PROGRAM CAN_comm
VAR
	i : INT := 0; // data 0 - 7 
	j : INT := 1; // coil 1-10
	k : INT := 1; // uc 1-10
	
	hmi_sendRequest : BOOL;
	hmi_step1 : BOOL;
	hmi_step2 : BOOL;
	hmi_step3 : BOOL;
	hmi_step4 : BOOL;
	hmi_step5 : BOOL;
	//hmi_CanTxB_str	: ARRAY [0..7] OF STRING;
	//hmi_CanTxB		: ARRAY [0..7] OF BYTE;
	hmi_CanTx_ID_str	: STRING;
	hmi_CanTx_ID		: UDINT;
	//hmi_CanTx_length	: UINT;
	hmi_CanTx_desiredID : STRING;
	hmi_CanTx_desID		: BYTE;

END_VAR

//0x0CF091 XX ELECTRICAL DATA
//0x0CF092 XX THERMAL DATA

//XX 
// ie 0x11[overvoltage][imbalance][blancing]
//data[0] = Electrical flag | data[1], data[2] = Voltage sum | data[3], data[4] = highest voltage | data[5], data[6] = average voltage | data[7] = life counter
//data[0].0
//data[0].1  Balancing
//data[0].2  
//data[0].3  Imbalance
//data[0].4
//data[0].5  Overvoltage
//data[0].6 = 1
//data[0].7 = 1

Devices.Coil[j].UC_Dummy_ID_hexstr :=  (DWORD_TO_HEXSTR (in := Devices.Coil[j].UltraCap_Dummy.R2_06_UC_Rx_cobID, iPrecision := 2, bLoCase := FALSE));
	//Devices.Coil[1].UltraCap_CAN_ID := Replace (STR1 := Devices.Coil[1].UltraCap_CAN_ID, '',1,1);
	//Devices.Coil[j].UltraCap_CAN_RxMsgNum[k].cobID := LEFT (Devices.Coil[j].UltraCap_CAN_RxMsgNum[k].cobID, 5);

(*	Devices.Coil[j].UltraCap_CAN_RxMsgNum[0].byteData_hexstr[0] := BYTE_TO_HEXSTR (in := Devices.Coil[j].UltraCap_CAN_RxMsg[0].data[0], iPrecision := 2, bLoCase := FALSE);
	Devices.Coil[j].UltraCap_CAN_RxMsgNum[0].byteData_hexstr[1] := BYTE_TO_HEXSTR (in := Devices.Coil[j].UltraCap_CAN_RxMsg[0].data[1], iPrecision := 2, bLoCase := FALSE);
	Devices.Coil[j].UltraCap_CAN_RxMsgNum[0].byteData_hexstr[2] := BYTE_TO_HEXSTR (in := Devices.Coil[j].UltraCap_CAN_RxMsg[0].data[2], iPrecision := 2, bLoCase := FALSE);
	Devices.Coil[j].UltraCap_CAN_RxMsgNum[0].byteData_hexstr[3] := BYTE_TO_HEXSTR (in := Devices.Coil[j].UltraCap_CAN_RxMsg[0].data[3], iPrecision := 2, bLoCase := FALSE);
	Devices.Coil[j].UltraCap_CAN_RxMsgNum[0].byteData_hexstr[4] := BYTE_TO_HEXSTR (in := Devices.Coil[j].UltraCap_CAN_RxMsg[0].data[4], iPrecision := 2, bLoCase := FALSE);
	Devices.Coil[j].UltraCap_CAN_RxMsgNum[0].byteData_hexstr[5] := BYTE_TO_HEXSTR (in := Devices.Coil[j].UltraCap_CAN_RxMsg[0].data[5], iPrecision := 2, bLoCase := FALSE);
	Devices.Coil[j].UltraCap_CAN_RxMsgNum[0].byteData_hexstr[6] := BYTE_TO_HEXSTR (in := Devices.Coil[j].UltraCap_CAN_RxMsg[0].data[6], iPrecision := 2, bLoCase := FALSE);
	Devices.Coil[j].UltraCap_CAN_RxMsgNum[0].byteData_hexstr[7] := BYTE_TO_HEXSTR (in := Devices.Coil[j].UltraCap_CAN_RxMsg[0].data[7], iPrecision := 2, bLoCase := FALSE);
	*)
	
FOR j := 1 TO 10 BY 1 DO 
	FOR k := 1 TO 10 BY 1 DO
		Devices.Coil[j].CapVoltage[k] := LREAL_TO_INT (Devices.Coil[j].UltraCap[k].Elec_VoltageSum);
		Devices.Coil[j].CapCellTemp[k] := LREAL_TO_INT (Devices.Coil[j].UltraCap[k].Therm_HighestCell); //sample the highest cell temperature
	END_FOR;
END_FOR;

//output set address for new UC - 7F 
//taking input from HMI
hmi_CanTx_ID := STRING_TO_UDINT (hmi_CanTx_ID_str);
hmi_CanTx_desID := STRING_TO_BYTE (hmi_CanTx_desiredID);
(*FOR i := 0 TO 7 BY 1 DO 
	hmi_CanTxB[i] := STRING_TO_BYTE (hmi_CanTxB_str[i]);
END_FOR;
	
IF hmi_sendRequest = TRUE THEN
	Devices.Coil[1].CanTx_config_ID := hmi_CanTx_ID;
	Devices.Coil[1].CanTx_config_length := hmi_CanTx_length;
	Devices.Coil[1].CanTx_config_request[0] := hmi_CanTxB[0];
	Devices.Coil[1].CanTx_config_request[1] := hmi_CanTxB[1];
	Devices.Coil[1].CanTx_config_request[2] := hmi_CanTxB[2];
	Devices.Coil[1].CanTx_config_request[3] := hmi_CanTxB[3];
	Devices.Coil[1].CanTx_config_request[4] := hmi_CanTxB[4];
ELSE 
	Devices.Coil[1].CanTx_config_ID := 16#00000000;
	Devices.Coil[1].CanTx_config_request[0] := 16#00;
	Devices.Coil[1].CanTx_config_request[1] := 16#00;
	Devices.Coil[1].CanTx_config_request[2] := 16#00;
	Devices.Coil[1].CanTx_config_request[3] := 16#00;
	Devices.Coil[1].CanTx_config_request[4] := 16#00;
	Devices.Coil[1].CanTx_config_request[5] := 16#00;
	Devices.Coil[1].CanTx_config_request[6] := 16#00;
	Devices.Coil[1].CanTx_config_request[7] := 16#00;
END_IF;
*)


IF hmi_step1 = TRUE THEN
	Devices.Coil[1].CanTx_config_ID := hmi_CanTx_ID;
	Devices.Coil[1].CanTx_config_length := 3;
	Devices.Coil[1].CanTx_config_request[0] := 16#02;
	Devices.Coil[1].CanTx_config_request[1] := 16#10;
	Devices.Coil[1].CanTx_config_request[2] := 16#03;
	
(*	Output.R2_06_CANrequest.cobId := 16#0CDA7FCC;
	Output.R2_06_CANrequest.length := 3;
	Output.R2_06_CANrequest.data[0] := 16#02;
	Output.R2_06_CANrequest.data[1] := 16#10;
	Output.R2_06_CANrequest.data[2] := 16#03;
	Output.R2_06_CANrequest.data[3] := 16#00;
	Output.R2_06_CANrequest.data[4] := 16#00;
	Output.R2_06_CANrequest.data[5] := 16#00;
	Output.R2_06_CANrequest.data[6] := 16#00;
	Output.R2_06_CANrequest.data[7] := 16#00;*)

ELSIF hmi_step2 = TRUE THEN
	Devices.Coil[1].CanTx_config_ID := hmi_CanTx_ID;
	Devices.Coil[1].CanTx_config_length := 3;
	Devices.Coil[1].CanTx_config_request[0] := 16#02;
	Devices.Coil[1].CanTx_config_request[1] := 16#27;
	Devices.Coil[1].CanTx_config_request[2] := 16#03;
	(*Output.R2_06_CANrequest.cobId := 16#0CDA7FCC;
	Output.R2_06_CANrequest.length := 3;
	Output.R2_06_CANrequest.data[0] := 16#02;
	Output.R2_06_CANrequest.data[1] := 16#27;
	Output.R2_06_CANrequest.data[2] := 16#01;
	Output.R2_06_CANrequest.data[3] := 16#00;
	Output.R2_06_CANrequest.data[4] := 16#00;
	Output.R2_06_CANrequest.data[5] := 16#00;
	Output.R2_06_CANrequest.data[6] := 16#00;
	Output.R2_06_CANrequest.data[7] := 16#00;
	*)
ELSIF hmi_step3 = TRUE THEN
	Devices.Coil[1].CanTx_config_ID := hmi_CanTx_ID;
	Devices.Coil[1].CanTx_config_length := 5;
	Devices.Coil[1].CanTx_config_request[0] := 16#04;
	Devices.Coil[1].CanTx_config_request[1] := 16#27;
	Devices.Coil[1].CanTx_config_request[2] := 16#02;
	Devices.Coil[1].CanTx_config_request[3] := 16#78;
	Devices.Coil[1].CanTx_config_request[4] := 16#9A;
	(*Output.R2_06_CANrequest.cobId := 16#0CDA7FCC;
	Output.R2_06_CANrequest.length := 5;
	Output.R2_06_CANrequest.data[0] := 16#04;
	Output.R2_06_CANrequest.data[1] := 16#27;
	Output.R2_06_CANrequest.data[2] := 16#02;
	Output.R2_06_CANrequest.data[3] := 16#78;
	Output.R2_06_CANrequest.data[4] := 16#9A;
	Output.R2_06_CANrequest.data[5] := 16#00;
	Output.R2_06_CANrequest.data[6] := 16#00;
	Output.R2_06_CANrequest.data[7] := 16#00;	
	*)
ELSIF hmi_step4 = TRUE THEN 
	Devices.Coil[1].CanTx_config_ID := hmi_CanTx_ID;
	Devices.Coil[1].CanTx_config_length := 5;
	Devices.Coil[1].CanTx_config_request[0] := 16#04;
	Devices.Coil[1].CanTx_config_request[1] := 16#2E;
	Devices.Coil[1].CanTx_config_request[2] := 16#FD;
	Devices.Coil[1].CanTx_config_request[3] := 16#08;
	Devices.Coil[1].CanTx_config_request[4] := hmi_CanTx_desID; //desirable cobID / device ID
	(*Output.R2_06_CANrequest.cobId := 16#0CDA7FCC;
	Output.R2_06_CANrequest.length := 5;
	Output.R2_06_CANrequest.data[0] := 16#04;
	Output.R2_06_CANrequest.data[1] := 16#2E;
	Output.R2_06_CANrequest.data[2] := 16#FD;
	Output.R2_06_CANrequest.data[3] := 16#08;
	Output.R2_06_CANrequest.data[4] := 16#02; //desirable cobID / device ID
	Output.R2_06_CANrequest.data[5] := 16#00;
	Output.R2_06_CANrequest.data[6] := 16#00;
	Output.R2_06_CANrequest.data[7] := 16#00;
	*)
ELSIF hmi_step5 = TRUE THEN 
	Devices.Coil[1].CanTx_config_ID := hmi_CanTx_ID;
	Devices.Coil[1].CanTx_config_length := 4;
	Devices.Coil[1].CanTx_config_request[0] := 16#03; //restart software
	Devices.Coil[1].CanTx_config_request[1] := 16#11;
	Devices.Coil[1].CanTx_config_request[2] := 16#01;
	Devices.Coil[1].CanTx_config_request[3] := 16#08;
	(*Output.R2_06_CANrequest.cobId:= 16#0CDA7FCC;
	Output.R2_06_CANrequest.length := 4;
	Output.R2_06_CANrequest.data[0] := 16#03;
	Output.R2_06_CANrequest.data[1] := 16#11;
	Output.R2_06_CANrequest.data[2] := 16#01;
	Output.R2_06_CANrequest.data[3] := 16#00;
	Output.R2_06_CANrequest.data[4] := 16#00;
	Output.R2_06_CANrequest.data[5] := 16#00;
	Output.R2_06_CANrequest.data[6] := 16#00;
	Output.R2_06_CANrequest.data[7] := 16#00;
	*)
ELSE 
	Devices.Coil[1].CanTx_config_ID := 16#00000000;
	Devices.Coil[1].CanTx_config_request[0] := 16#00;
	Devices.Coil[1].CanTx_config_request[1] := 16#00;
	Devices.Coil[1].CanTx_config_request[2] := 16#00;
	Devices.Coil[1].CanTx_config_request[3] := 16#00;
	Devices.Coil[1].CanTx_config_request[4] := 16#00;
	Devices.Coil[1].CanTx_config_request[5] := 16#00;
	Devices.Coil[1].CanTx_config_request[6] := 16#00;
	Devices.Coil[1].CanTx_config_request[7] := 16#00;
END_IF;


IF i > 7 THEN
	i := 0;
END_IF;

IF j > 10 THEN
	j := 1;
END_IF;

IF k > 10 THEN
	k := 1;
END_IF;

END_PROGRAM

(* stored: Version 1.1.0.1, ProductVersion 3.1.4024.11
   POU CAN_comm: Id {3e952c50-c200-4586-9bea-34a28232d4e5}, SpecialFunc None *)
